// TIA Portal project "Farol_Patio" (V15)

(* hardware
DEVICE "S7-1200 station_1"  S7-1200 Station
   slot 0: "Rack_0"  S7-1200 Rack  Rack  V1.0
   slot 1: "PLC_1"  CPU 1214C DC/DC/DC  6ES7 214-1AG40-0XB0  V4.2
*)

// ===== PLC "PLC_1"  CPU 1214C DC/DC/DC =====

VAR_GLOBAL   // PLC tag table "Default tag table"
   "DI_Botao_Pedestre" AT %I0.0 : Bool;
   "DI_Botao_Pedestre_1" AT %I0.1 : Bool;
   "DO_Verde_P" AT %Q0.0 : Bool;
   "DO_Vermelho_P" AT %Q0.4 : Bool;
   "DO_Verde_C" AT %Q0.5 : Bool;
   "DO_Vermelho_C" AT %Q0.3 : Bool;
   "M_Horario_Parada" AT %M2.1 : Bool;
   "TimeOfDay" AT %MD2 : Time_Of_Day;
END_VAR

VAR_GLOBAL   // PLC tag table "ClockMemories"
   "Clock_Byte" AT %MB0 : Byte;
   "Clock_10Hz" AT %M0.0 : Bool;
   "Clock_5Hz" AT %M0.1 : Bool;
   "Clock_2.5Hz" AT %M0.2 : Bool;
   "Clock_2Hz" AT %M0.3 : Bool;
   "Clock_1.25Hz" AT %M0.4 : Bool;
   "Clock_1Hz" AT %M0.5 : Bool;
   "Clock_0.625Hz" AT %M0.6 : Bool;
   "Clock_0.5Hz" AT %M0.7 : Bool;
   "System_Byte" AT %MB1 : Byte;
   "FirstScan" AT %M1.0 : Bool;
   "DiagStatusUpdate" AT %M1.1 : Bool;
   "AlwaysTRUE" AT %M1.2 : Bool;
   "AlwaysFALSE" AT %M1.3 : Bool;
END_VAR

DATA_BLOCK "Lunch_Time_DB"   // DB2
{ S7_Optimized_Access := 'TRUE' }
VERSION : 0.1
// stored: InstanceOfName Lunch_Time
"Lunch_Time"
BEGIN
END_DATA_BLOCK

DATA_BLOCK "Humble_With_ControlTower_DB"   // DB3
{ S7_Optimized_Access := 'TRUE' }
VERSION : 0.1
// stored: InstanceOfName Humble_With_ControlTower
"Humble_With_ControlTower"
BEGIN
END_DATA_BLOCK

DATA_BLOCK "GeneralMemories"   // DB7
{ S7_Optimized_Access := 'TRUE' }
VERSION : 0.1
   VAR
      Inputs : Struct
         Botão_Pedestre : Bool;
         Botão_Pedestre_1 : Bool;
      END_STRUCT;
      Outputs : Struct
         VerdeP : Bool;
         VermelhoP : Bool;
         VerdeC : Bool;
         VermelhoC : Bool;
      END_STRUCT;
   END_VAR
BEGIN
END_DATA_BLOCK

DATA_BLOCK "FB10_Farol_DB"   // DB8
{ S7_Optimized_Access := 'FALSE' }
VERSION : 0.1
// stored: InstanceOfName FB10_Farol
"FB10_Farol"
BEGIN
END_DATA_BLOCK

FUNCTION_BLOCK "Lunch_Time"   // FB1, LAD
{ S7_Optimized_Access := 'TRUE' }
VERSION : 0.1
   VAR_OUTPUT
      OUT_Time_of_day : Time_Of_Day;
      OUT_HorarioParada : Bool;
   END_VAR
   VAR
      S_Out_ReadTimeSystem : DTL;
      S_OutReadConvert : DTL;
      S_Return_Value : Int;
      S_Actual : Time_Of_Day;
      S_HorarioParada : Bool;
      S_HorarioParada_1 : Bool;
      S_HorarioParada_2 : Bool;
      S_HorarioParada_3 : Bool;
      S_HorarioParada_4 : Bool;
   END_VAR
   VAR CONSTANT
      S_BreakFastStarts : Time_Of_Day := TOD#06:30:00;
      S_BreakFastStop : Time_Of_Day := TOD#07:05:00;
      S_LunchTimeStart : Time_Of_Day := TOD#11:00:00;
      S_LunchTimeStop : Time_Of_Day := TOD#12:30:00;
      S_ExitTimeStart : Time_Of_Day := TOD#15:45:00;
      S_ExitTimeStop : Time_Of_Day := TOD#16:30:00;
      S_DinnerStart : Time_Of_Day := TOD#21:00:00;
      S_DinnerStop : Time_Of_Day := TOD#22:00:00;
      S_ExitTimeStart_2 : Time_Of_Day := TOD#23:50:00;
      S_ExitTimeStop_2 : Time_Of_Day := TOD#00:20:00;
   END_VAR
BEGIN

REGION Network 1: Pega a hora do sistema e Sub trai um valor
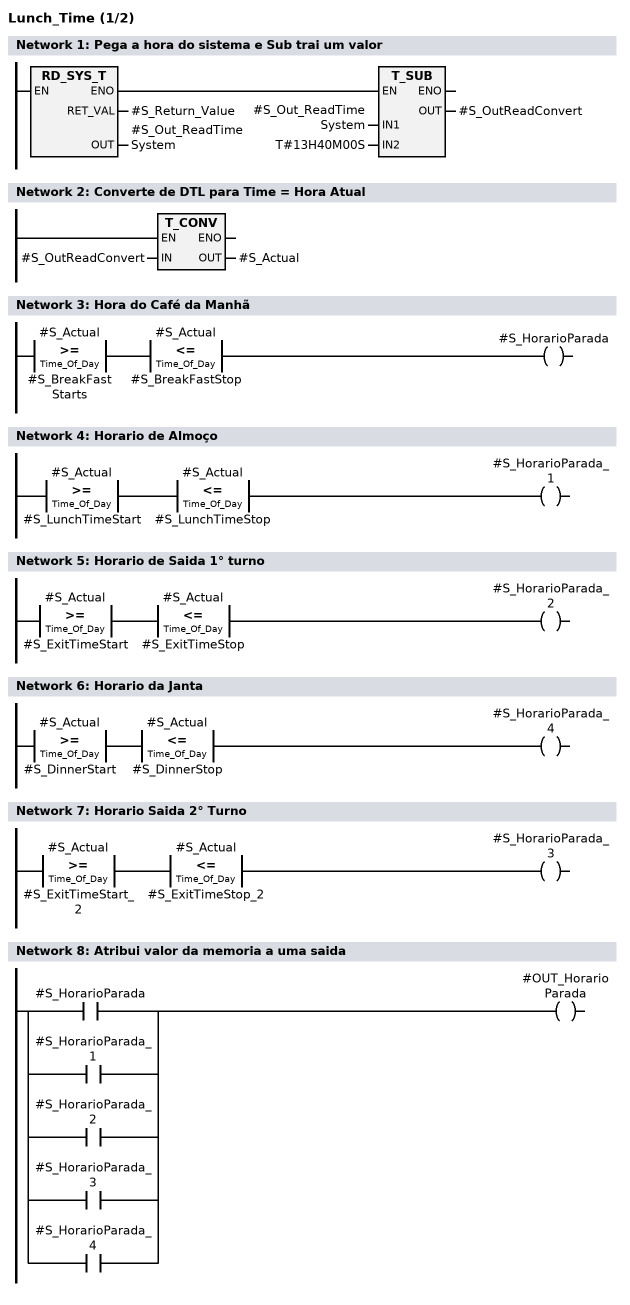
   // ENO of a box is taken as its EN; it also drops when the box reports an error
   #S_Return_Value := RD_SYS_T(OUT => #S_Out_ReadTimeSystem);
   #S_OutReadConvert := T_SUB(IN1 := #S_Out_ReadTimeSystem, IN2 := T#13H40M00S);
END_REGION

REGION Network 2: Converte de DTL para Time = Hora Atual
   #S_Actual := T_CONV(IN := #S_OutReadConvert);
END_REGION

REGION Network 3: Hora do Café da Manhã
   RUNG wire#powerrail
      { S7_Templates := "SrcType := Time_Of_Day" } GE_Contact(in1 := #S_Actual, in2 := #S_BreakFastStarts)
      { S7_Templates := "SrcType := Time_Of_Day" } LE_Contact(in1 := #S_Actual, in2 := #S_BreakFastStop)
      Coil( #S_HorarioParada )
   END_RUNG
   // the same network as SCL:
   #S_HorarioParada := (#S_Actual >= #S_BreakFastStarts) AND (#S_Actual <= #S_BreakFastStop);
END_REGION

REGION Network 4: Horario de Almoço
   RUNG wire#powerrail
      { S7_Templates := "SrcType := Time_Of_Day" } GE_Contact(in1 := #S_Actual, in2 := #S_LunchTimeStart)
      { S7_Templates := "SrcType := Time_Of_Day" } LE_Contact(in1 := #S_Actual, in2 := #S_LunchTimeStop)
      Coil( #S_HorarioParada_1 )
   END_RUNG
   // the same network as SCL:
   #S_HorarioParada_1 := (#S_Actual >= #S_LunchTimeStart) AND (#S_Actual <= #S_LunchTimeStop);
END_REGION

REGION Network 5: Horario de Saida 1° turno
   RUNG wire#powerrail
      { S7_Templates := "SrcType := Time_Of_Day" } GE_Contact(in1 := #S_Actual, in2 := #S_ExitTimeStart)
      { S7_Templates := "SrcType := Time_Of_Day" } LE_Contact(in1 := #S_Actual, in2 := #S_ExitTimeStop)
      Coil( #S_HorarioParada_2 )
   END_RUNG
   // the same network as SCL:
   #S_HorarioParada_2 := (#S_Actual >= #S_ExitTimeStart) AND (#S_Actual <= #S_ExitTimeStop);
END_REGION

REGION Network 6: Horario da Janta
   RUNG wire#powerrail
      { S7_Templates := "SrcType := Time_Of_Day" } GE_Contact(in1 := #S_Actual, in2 := #S_DinnerStart)
      { S7_Templates := "SrcType := Time_Of_Day" } LE_Contact(in1 := #S_Actual, in2 := #S_DinnerStop)
      Coil( #S_HorarioParada_4 )
   END_RUNG
   // the same network as SCL:
   #S_HorarioParada_4 := (#S_Actual >= #S_DinnerStart) AND (#S_Actual <= #S_DinnerStop);
END_REGION

REGION Network 7: Horario Saida 2° Turno
   RUNG wire#powerrail
      { S7_Templates := "SrcType := Time_Of_Day" } GE_Contact(in1 := #S_Actual, in2 := #S_ExitTimeStart_2)
      { S7_Templates := "SrcType := Time_Of_Day" } LE_Contact(in1 := #S_Actual, in2 := #S_ExitTimeStop_2)
      Coil( #S_HorarioParada_3 )
   END_RUNG
   // the same network as SCL:
   #S_HorarioParada_3 := (#S_Actual >= #S_ExitTimeStart_2) AND (#S_Actual <= #S_ExitTimeStop_2);
END_REGION

REGION Network 8: Atribui valor da memoria a uma saida
   RUNG wire#powerrail
      Contact( #S_HorarioParada )
      wire#w1
      Coil( #OUT_HorarioParada )
   END_RUNG
   RUNG wire#powerrail
      Contact( #S_HorarioParada_1 )
   END_RUNG wire#w1
   RUNG wire#powerrail
      Contact( #S_HorarioParada_2 )
   END_RUNG wire#w1
   RUNG wire#powerrail
      Contact( #S_HorarioParada_3 )
   END_RUNG wire#w1
   RUNG wire#powerrail
      Contact( #S_HorarioParada_4 )
   END_RUNG wire#w1
   // the same network as SCL:
   #OUT_HorarioParada := #S_HorarioParada OR #S_HorarioParada_1 OR #S_HorarioParada_2 OR #S_HorarioParada_3 OR #S_HorarioParada_4;
END_REGION

REGION Network 9
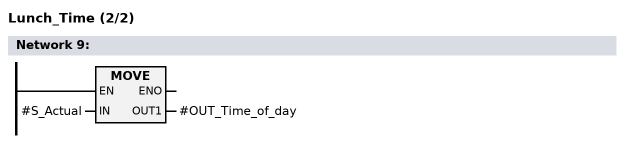
   RUNG wire#powerrail
      Move(in := #S_Actual, out1 => #OUT_Time_of_day)
   END_RUNG
   // the same network as SCL:
   #OUT_Time_of_day := #S_Actual;
END_REGION
END_FUNCTION_BLOCK

FUNCTION_BLOCK "Humble_With_ControlTower"   // FB3, LAD
{ S7_Optimized_Access := 'TRUE' }
VERSION : 0.1
BEGIN
END_FUNCTION_BLOCK

FUNCTION_BLOCK "FB10_Farol"   // FB4, SCL
{ S7_Optimized_Access := 'FALSE' }
VERSION : 0.1
   VAR_INPUT
      "IN_Libera.Pedestre" : Bool;   // Sinal do botão para liberar o pedestre.
      "IN_Clock.1s" : Bool;   // Sinal do Clock Memory de um segundo.
      IN_Horario_Parada : Bool;
   END_VAR
   VAR_OUTPUT
      "OUT_Verde.Pedestre" : Bool;   // Lâmpada do Farol "Verde" Pedestre.
      "OUT_Vermelho.Pedestre" : Bool;   // Lâmpada do Farol "Vermelho" Pedestre.
      "OUT_Verde.Caminhao" : Bool;   // Lâmpada do Farol "Verde" Caminhão.
      "OUT_Vermelho.Caminhao" : Bool;   // Lâmpada do Farol "Vermelho" Caminhão.
   END_VAR
   VAR
      TIMER_Farol : TON_TIME;   // Temporizador para as sequencias do farol.
      "MS_Timer_Farol.IN" : Bool;   // Memória Statica para start do temporizador Timer farol.
      MS_Sequencia : Int;   // Memória Statica para atribuir as sequencias.
      "MS_Sequencia.2" : Bool;   // Memória Statica para lógica da sequencia 2.
      "MS_Libera.Pedestre" : Bool;   // Memória Statica para Lógica de acionamento do botão libera pedestre.
      "MS_Verde.Pedestre" : Bool;   // Memória Statica para lógica de acionamento da saída (Lâmpada do Farol "Verde" Pedestre).
      "MS_Vermelho.Pedestre" : Bool;   // Memória Statica para lógica de acionamento da saída (Lâmpada do Farol "Vermelho" Pedestre).
      "MS_Verde.Caminhao" : Bool;   // Memória Statica para lógica de acionamento da saída (Lâmpada do Farol "Verde" Caminhão).
      "MS_Vermelho.Caminhao" : Bool;   // Memória Statica para lógica de acionamento da saída (Lâmpada do Farol "Vermelho" Caminhão).
      MS_Out_ReadTime : DTL;
      MS_ReturnValRDST : Int;
      MS_HorarioParada : Bool;
   END_VAR
BEGIN
   // GOD BE PRAISED

   // LÓGICA DE COMANDO PARA SEQUENCIA (1).
   #MS_HorarioParada := #IN_Horario_Parada;

   // Se o botão de libera pedestre não for acionado, a variavel "sequencia" executa a (sequencia 1).

   IF NOT #"MS_Libera.Pedestre" AND NOT #MS_HorarioParada THEN
       #MS_Sequencia := 1;
   END_IF;
   //~~~~~~~~~~~~~~~~~~~~~~~~~~~~~~~~~~~~~~~~~~~~~~~~~~~~~~~~~~~~~~~~~~~~~~~~~~~~~~~~~~~~~~~~~~~~~~~~~~~~~~~~~~~~~~~~~~~~~~~~~~~~~~~~~~~~~~~~~~~~~~~~~

   // ACIONAMENTO DO BOTÃO "LIBERA PEDESTRE".

   // Se o botão "Libera.Pedestre" for acionado, a memoria stática "MS_Libera.Pedestre" é acionada.

   IF #"IN_Libera.Pedestre" AND NOT #MS_HorarioParada  THEN
       #"MS_Libera.Pedestre" := 1;
   END_IF;

   //~~~~~~~~~~~~~~~~~~~~~~~~~~~~~~~~~~~~~~~~~~~~~~~~~~~~~~~~~~~~~~~~~~~~~~~~~~~~~~~~~~~~~~~~~~~~~~~~~~~~~~~~~~~~~~~~~~~~~~~~~~~~~~~~~~~~~~~~~~~~~~~~~

   // ACIONAMENTO DA CONTAGEM DO TIMER DO FAROL.

   // Quando a memoria statica "MS_Libera.Pedestre" é acionada, o timer do Farol é iniciado.

   #"MS_Timer_Farol.IN" := #"MS_Libera.Pedestre";
   //~~~~~~~~~~~~~~~~~~~~~~~~~~~~~~~~~~~~~~~~~~~~~~~~~~~~~~~~~~~~~~~~~~~~~~~~~~~~~~~~~~~~~~~~~~~~~~~~~~~~~~~~~~~~~~~~~~~~~~~~~~~~~~~~~~~~~~~~~~~~~~~~~

   // LÓGICA DE COMANDO PARA SEQUENCIA (2).

   // Se a memoria statica #"MS_Libera.Pedestre" estiver acionada e a memoria statica #"MS_Sequencia.2" não estiver acionada,
   //a variavel "sequencia" executa a (sequencia 2).

   IF #"MS_Libera.Pedestre" AND
       NOT #"MS_Sequencia.2" THEN
       #MS_Sequencia := 2;
   END_IF;
   //~~~~~~~~~~~~~~~~~~~~~~~~~~~~~~~~~~~~~~~~~~~~~~~~~~~~~~~~~~~~~~~~~~~~~~~~~~~~~~~~~~~~~~~~~~~~~~~~~~~~~~~~~~~~~~~~~~~~~~~~~~~~~~~~~~~~~~~~~~~~~~~~~

   // LÓGICA DE COMANDO PARA SEQUENCIA (3).

   // Quando o Timer do farol ultrapassar 10s, e contar até 85s, a memoria statica #"MS_Sequencia.2" ira acionar e cortar a (sequencia 2),
   //e a variavel "sequencia" executa a (sequencia 3).

   IF (#TIMER_Farol.ET > T#10s) AND
       (#TIMER_Farol.ET <= T#85s) THEN
       #"MS_Sequencia.2" := 1;
       #MS_Sequencia := 3;


   END_IF;
   //~~~~~~~~~~~~~~~~~~~~~~~~~~~~~~~~~~~~~~~~~~~~~~~~~~~~~~~~~~~~~~~~~~~~~~~~~~~~~~~~~~~~~~~~~~~~~~~~~~~~~~~~~~~~~~~~~~~~~~~~~~~~~~~~~~~~~~~~~~~~~~~~~

   // LÓGICA DE COMANDO PARA SEQUENCIA (4).

   // Quando o Timer do farol ultrapassar 85s, a variavel "sequencia" executa a (sequencia 4).

   IF (#TIMER_Farol.ET > T#85s) THEN
       #MS_Sequencia := 4;
   END_IF;
   //~~~~~~~~~~~~~~~~~~~~~~~~~~~~~~~~~~~~~~~~~~~~~~~~~~~~~~~~~~~~~~~~~~~~~~~~~~~~~~~~~~~~~~~~~~~~~~~~~~~~~~~~~~~~~~~~~~~~~~~~~~~~~~~~~~~~~~~~~~~~~~~~~

   // LÓGICA PARA RETORNAR PARA SEQUENCIA 1.

   // Quando o Timer do farol chegar no final da contagem, a memoria statica #"MS_Libera.Pedestre" é desligada junto com a memoria
   // #"MS_Sequencia.2" fazendo a variavel "sequencia" executar a (sequencia 1) novamente.

   IF #TIMER_Farol.Q THEN
       #"MS_Libera.Pedestre" := 0;
       #"MS_Sequencia.2" := 0;
   END_IF;
   //~~~~~~~~~~~~~~~~~~~~~~~~~~~~~~~~~~~~~~~~~~~~~~~~~~~~~~~~~~~~~~~~~~~~~~~~~~~~~~~~~~~~~~~~~~~~~~~~~~~~~~~~~~~~~~~~~~~~~~~~~~~~~~~~~~~~~~~~~~~~~~~~~

   // TIMER DO FAROL.

   // O temporizador "Timer farol" conta todo o tempo necessário para as sequecias, e para cada tempo individual da sequencia, é
   // trabalhado com largura de tempo.

   #TIMER_Farol(IN := #"MS_Timer_Farol.IN",
                PT := T#95s);
   //~~~~~~~~~~~~~~~~~~~~~~~~~~~~~~~~~~~~~~~~~~~~~~~~~~~~~~~~~~~~~~~~~~~~~~~~~~~~~~~~~~~~~~~~~~~~~~~~~~~~~~~~~~~~~~~~~~~~~~~~~~~~~~~~~~~~~~~~~~~~~~~~~
   // Logica de comando Horario de Parada
   IF #MS_HorarioParada THEN
       #MS_Sequencia := 5;
       ;
   END_IF;

   // FUNÇÃO PARA EXECUTAR A AÇÃO CONFORME SEQUENCIA ATRIBUIDA.

   // Ao mudar o valor da variavel "#MS_Sequencia" o programa executa uma função diferente de acordo programado.

   CASE #MS_Sequencia OF


       1:  // Lógica de acionamento para sequencia 1.

           #"MS_Verde.Pedestre" := 0;
           #"MS_Vermelho.Pedestre" := 1;
           #"MS_Verde.Caminhao" := 1;
           #"MS_Vermelho.Caminhao" := 0;

       2:  // Lógica de acionamento para sequencia 2.

           #"MS_Verde.Pedestre" := 0;
           #"MS_Vermelho.Pedestre" := 1;
           #"MS_Verde.Caminhao" := 0;
           #"MS_Vermelho.Caminhao" := #"IN_Clock.1s";

       3:  // Lógica de acionamento para sequencia 3.

           #"MS_Verde.Pedestre" := 1;
           #"MS_Vermelho.Pedestre" := 0;
           #"MS_Verde.Caminhao" := 0;
           #"MS_Vermelho.Caminhao" := 1;

       4:  // Lógica de acionamento para sequencia 4.

           #"MS_Verde.Pedestre" := 0;
           #"MS_Vermelho.Pedestre" := #"IN_Clock.1s";
           #"MS_Verde.Caminhao" := 0;
           #"MS_Vermelho.Caminhao" := 1;
       5:
           #"MS_Verde.Pedestre" := 1;
           #"MS_Vermelho.Pedestre" := 0;
           #"MS_Verde.Caminhao" := 0;
           #"MS_Vermelho.Caminhao" := 1; ;


   END_CASE;







   // ATRIBUIÇÃO PARA AS SAÍDAS.

   #"OUT_Verde.Pedestre" := #"MS_Verde.Pedestre";
   #"OUT_Vermelho.Pedestre" := #"MS_Vermelho.Pedestre";
   #"OUT_Verde.Caminhao" := #"MS_Verde.Caminhao";
   #"OUT_Vermelho.Caminhao" := #"MS_Vermelho.Caminhao";
END_FUNCTION_BLOCK

FUNCTION "General.Memories" : Void   // FC1, SCL
{ S7_Optimized_Access := 'TRUE' }
VERSION : 0.1
   VAR_INPUT
      IN_Botão_Pedestre : Bool;
      IN_Botão_Pedestre_1 : Bool;
      IN_VerdeP : Bool;
      IN_VermelhoP : Bool;
      IN_VerdeC : Bool;
      IN_VermelhoC : Bool;
   END_VAR
   VAR_OUTPUT
      OUT_Botão_Pedestre : Bool;
      OUT_Botão_Pedestre_1 : Bool;
      OUT_VerdeP : Bool;
      OUT_VermelhoP : Bool;
      OUT_VerdeC : Bool;
      OUT_VermelhoC : Bool;
   END_VAR
BEGIN


   #OUT_Botão_Pedestre := #IN_Botão_Pedestre OR #IN_Botão_Pedestre_1;
   #OUT_Botão_Pedestre_1 := #IN_Botão_Pedestre_1;
   #OUT_VerdeP := #IN_VerdeP;
   #OUT_VermelhoP := #IN_VermelhoP;
   #OUT_VerdeC := #IN_VerdeC;
   #OUT_VermelhoC := #IN_VermelhoC;
END_FUNCTION

ORGANIZATION_BLOCK "Main"   // OB1, LAD, ProgramCycle
TITLE = "Main Program Sweep (Cycle)"
{ S7_Optimized_Access := 'TRUE' }
VERSION : 0.1
   VAR_INPUT
      Initial_Call : Bool;   // Initial call of this OB
      Remanence : Bool;   // =True, if remanent data are available
   END_VAR
BEGIN

REGION Network 1
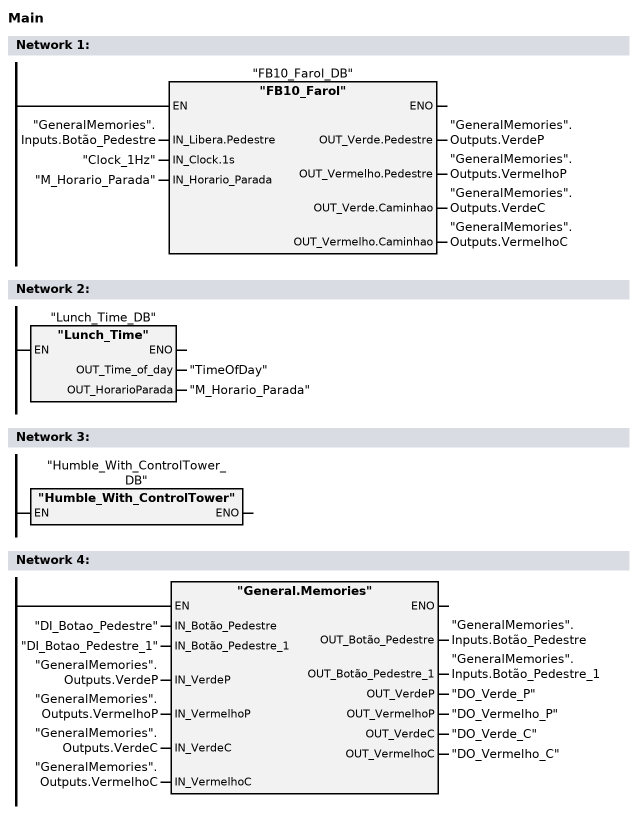
   RUNG wire#powerrail
      "FB10_Farol_DB"("IN_Libera.Pedestre" := "GeneralMemories".Inputs.Botão_Pedestre, "IN_Clock.1s" := "Clock_1Hz", IN_Horario_Parada := "M_Horario_Parada", "OUT_Verde.Pedestre" => "GeneralMemories".Outputs.VerdeP, "OUT_Vermelho.Pedestre" => "GeneralMemories".Outputs.VermelhoP, "OUT_Verde.Caminhao" => "GeneralMemories".Outputs.VerdeC, "OUT_Vermelho.Caminhao" => "GeneralMemories".Outputs.VermelhoC)
   END_RUNG
   // the same network as SCL:
   "FB10_Farol_DB"("IN_Libera.Pedestre" := "GeneralMemories".Inputs.Botão_Pedestre,   // "FB10_Farol"
                   "IN_Clock.1s" := "Clock_1Hz",
                   IN_Horario_Parada := "M_Horario_Parada",
                   "OUT_Verde.Pedestre" => "GeneralMemories".Outputs.VerdeP,
                   "OUT_Vermelho.Pedestre" => "GeneralMemories".Outputs.VermelhoP,
                   "OUT_Verde.Caminhao" => "GeneralMemories".Outputs.VerdeC,
                   "OUT_Vermelho.Caminhao" => "GeneralMemories".Outputs.VermelhoC);
END_REGION

REGION Network 2
   RUNG wire#powerrail
      "Lunch_Time_DB"(OUT_Time_of_day => "TimeOfDay", OUT_HorarioParada => "M_Horario_Parada")
   END_RUNG
   // the same network as SCL:
   "Lunch_Time_DB"(OUT_Time_of_day => "TimeOfDay", OUT_HorarioParada => "M_Horario_Parada");   // "Lunch_Time"
END_REGION

REGION Network 3
   RUNG wire#powerrail
      "Humble_With_ControlTower_DB"()
   END_RUNG
   // the same network as SCL:
   "Humble_With_ControlTower_DB"();   // "Humble_With_ControlTower"
END_REGION

REGION Network 4
   RUNG wire#powerrail
      "General.Memories"(IN_Botão_Pedestre := "DI_Botao_Pedestre", IN_Botão_Pedestre_1 := "DI_Botao_Pedestre_1", IN_VerdeP := "GeneralMemories".Outputs.VerdeP, IN_VermelhoP := "GeneralMemories".Outputs.VermelhoP, IN_VerdeC := "GeneralMemories".Outputs.VerdeC, IN_VermelhoC := "GeneralMemories".Outputs.VermelhoC, OUT_Botão_Pedestre => "GeneralMemories".Inputs.Botão_Pedestre, OUT_Botão_Pedestre_1 => "GeneralMemories".Inputs.Botão_Pedestre_1, OUT_VerdeP => "DO_Verde_P", OUT_VermelhoP => "DO_Vermelho_P", OUT_VerdeC => "DO_Verde_C", OUT_VermelhoC => "DO_Vermelho_C")
   END_RUNG
   // the same network as SCL:
   "General.Memories"(IN_Botão_Pedestre := "DI_Botao_Pedestre",
                      IN_Botão_Pedestre_1 := "DI_Botao_Pedestre_1",
                      IN_VerdeP := "GeneralMemories".Outputs.VerdeP,
                      IN_VermelhoP := "GeneralMemories".Outputs.VermelhoP,
                      IN_VerdeC := "GeneralMemories".Outputs.VerdeC,
                      IN_VermelhoC := "GeneralMemories".Outputs.VermelhoC,
                      OUT_Botão_Pedestre => "GeneralMemories".Inputs.Botão_Pedestre,
                      OUT_Botão_Pedestre_1 => "GeneralMemories".Inputs.Botão_Pedestre_1,
                      OUT_VerdeP => "DO_Verde_P",
                      OUT_VermelhoP => "DO_Vermelho_P",
                      OUT_VerdeC => "DO_Verde_C",
                      OUT_VermelhoC => "DO_Vermelho_C");
END_REGION
END_ORGANIZATION_BLOCK